Universal Robots PolyScope program: skrewdriving.urp

Program skrewdriving (installation=default directory=/home/ur/ursim-current/programs createdIn=5.14.0 lastSavedIn=5.13.0 robotSerialNumber=20195299999)
Calibrated DH parameters: a=[0, -0.6127, -0.57155, 0, 0, 0]; d=[0.1807, 0, 0, 0.17415, 0.11985, 0.11655]; alpha=[1.570796, 0, 0, 1.570796, -1.570796, 0]; deltaTheta=[0, 0, 0, 0, 0, 0]
InitVariablesNode
BeforeStart
  start_task := False
  'Define p1, p2, p3, p4, p5, p6 as Installation Variables'
  positions := [p1, p2, p3, p4, p5, p6, p7, p8]
  i := 0
Robot Program (runOnlyOnce=false)
  URCap HMI (Robpod HMI URcap, Robpod Cloud) dataModel(robpod.hmi.selected=/home/ur/ursim-current/programs/skrewdriving.hmi)
  Wait Condition expression=start_task
  i := 0
  Loop Counting (count=8) loopVariable(name=Loop_1)
    skrew_pose := positions[i]
    approach_pose := pose_trans(skrew_pose, p[0, 0, -skrew_length * 2 / 1000, 0, 0, 0])
    MoveL speed 250 mm/s, acceleration 1200 mm/s^2 (useActiveTCP=true) feature=Base
      Waypoint Variable (Variable): variable=approach_pose
      Waypoint Variable (Variable): variable=skrew_pose
    Set DigitalOutput pin=digital_out[1]; digitalValue=1
    Wait Sleep waitTime=2
    Set DigitalOutput pin=digital_out[1]; digitalValue=0
    MoveL speed 250 mm/s, acceleration 1200 mm/s^2 (useActiveTCP=true) feature=Base
      Waypoint Variable (Variable): variable=approach_pose
    i := i + 1
  start_task := False
